// Fluent builder interface for composing log entries.
// Obtain an instance via F_Log() or FB_Log.Log(), chain methods, and call CreateLog() to emit.
INTERFACE I_Logger

// Finalizes and sends the log entry. Must be called to emit the log.
// After CreateLog(), the builder is consumed — do not reuse without a new F_Log() call.
METHOD CreateLog
END_METHOD

// Adds a log argument. Supports all IEC 61131-3 types (BOOL, INT, REAL, STRING, etc.).
// Arguments are referenced by position in the message template: '{0}', '{1}', ...
// Values are serialized immediately — safe to call in loops with changing variables.
METHOD WithAnyArg : I_Logger
VAR_INPUT
	stArg		: ANY;
END_VAR
END_METHOD

(*
:Description: Bind this log entry to a specific FB_Span for explicit
trace context correlation.

When WithSpan is called, the log message will be associated with the span's
trace_id and span_id in the tc-otel backend, creating an explicit link in
the trace timeline.

Call before CreateLog to take effect. Calling after CreateLog has no effect.

Typical usage:

.. code-block:: pascal

    VAR
        spn : FB_Span;
    END_VAR

    F_Log(E_LogLevel.eInfo, 'operation started')
        .WithSpan(spn)
        .CreateLog();
*)
METHOD PUBLIC WithSpan : I_Logger
VAR_IN_OUT
	span : FB_Span;
END_VAR
END_METHOD

// Adds a pre-typed argument (T_Arg from Tc2_Utilities).
// Prefer WithAnyArg for most cases. WithTArg is for compatibility with Tc2 formatting functions.
METHOD INTERNAL WithTArg : I_Logger
VAR_INPUT
	stArg		: T_Arg;
END_VAR
END_METHOD

END_INTERFACE

(* stored: Version 1.1.0.1, ProductVersion 3.1.4026.18
   Itf I_Logger: Id {8b7a3ede-9c91-0d75-34fd-1cfbab5e4360}
   Method CreateLog: Id {c36020e1-7629-0123-1b40-b63c6b460407}
   Method WithAnyArg: Id {555dd333-7171-0d36-075f-37b8e2570086}
   Method WithSpan: Id {eefac63a-7e1f-0e5b-2261-2143375d8616}
   Method WithTArg: Id {d5ace616-21ca-09f8-328c-30dbd866d03e} *)
